# EPICS substitutions: ucmApp/Db/undulator/useg-poly-bb.substitutions
file poly-inpcp.template{
  pattern { OUTPUT , COEF0, COEF1, COEF2, COEF3, COEF4, COEF5, INPUT         , SCAN       , NAME}
          { I1XBBRAW , $(U):POLYI1XBB_A, $(U):POLYI1XBB_B , $(U):POLYI1XBB_C, $(U):POLYI1XBB_D, $(U):POLYI1XBB_E, $(U):POLYI1XBB_F, XACTNEGATIVE, "10 second",POLYI1XBB}
          { I1YBBRAW , $(U):POLYI1YBB_A, $(U):POLYI1YBB_B, $(U):POLYI1YBB_C, $(U):POLYI1YBB_D, $(U):POLYI1YBB_E, $(U):POLYI1YBB_F, XACTNEGATIVE, "10 second",POLYI1YBB}
          { I1XBBMMFL , $(U):POLYI1XBB_A, $(U):POLYI1XBB_B , $(U):POLYI1XBB_C, $(U):POLYI1XBB_D, $(U):POLYI1XBB_E, $(U):POLYI1XBB_F, XMMFL_NEG, "Passive",POLYI1XBBMMFL}
          { I1YBBMMFL , $(U):POLYI1YBB_A, $(U):POLYI1YBB_B, $(U):POLYI1YBB_C, $(U):POLYI1YBB_D, $(U):POLYI1YBB_E, $(U):POLYI1YBB_F, XMMFL_NEG, "Passive", POLYI1YBBMMFL}
          { I1XBB_BBA , $(U):POLYI1XBB_A, $(U):POLYI1XBB_B , $(U):POLYI1XBB_C, $(U):POLYI1XBB_D, $(U):POLYI1XBB_E, $(U):POLYI1XBB_F, LAST_BBA_NEG, "Passive",POLYI1XBBBBA}
          { I1YBB_BBA , $(U):POLYI1YBB_A, $(U):POLYI1YBB_B, $(U):POLYI1YBB_C, $(U):POLYI1YBB_D, $(U):POLYI1YBB_E, $(U):POLYI1YBB_F, LAST_BBA_NEG, "Passive", POLYI1YBBBBA}
}
